// TwinCAT 3 PLC project Tc_EvenLogger
// Title: Tc_SystemServices
// Company: NewEngineer
// Author: https://github.com/phucpha
// ProjectVersion: 0.0.0.1
// Description: This library use for AlarmControler, Recipemanager,..
// ProgramVersion: 3.1.4024.0
// libraries:
//   Recipe Management, * (System)
//   Tc2_Standard, * (Beckhoff Automation GmbH)
//   Tc2_System, * (Beckhoff Automation GmbH)
//   Tc2_Utilities, * (Beckhoff Automation GmbH)
//   Tc3_EventLogger, * (Beckhoff Automation GmbH)
//   Tc3_Module, * (Beckhoff Automation GmbH)
//   TC3_Utilities_C, * (NewEngineer)
//   VisuDialogs, * (System)
//   VisuSymbols,3.5.10.0,System
// project tree:
//   DUTs/AlarmsEventLogger/AlarmControler/ E_AlarmControlerState.TcDUT (not stored)
//   DUTs/AlarmsEventLogger/VisuEvents/ E_EventType.TcDUT (not stored), ST_BaseEvent.TcDUT (not stored), ST_Event.TcDUT (not stored)
//   DUTs/Recipe Manager/ E_RecipesManagerReturns.TcDUT (not stored), E_RecipesManagerState.TcDUT (not stored), E_RecipesManagerStateBackup.TcDUT (not stored), E_RecipesManagerStateCreateRemove.TcDUT (not stored), E_RecipesManagerStateInit.TcDUT (not stored), E_RecipesManagerStateReload.TcDUT (not stored)
//   DUTs/Visus/AlarmControl/ E_VisuCtrlAlarmControlState.TcDUT (not stored)
//   DUTs/Visus/RecipeManager/ E_VisuCtrlRecipeParameterType.TcDUT (not stored), E_VisuCtrlRecipesManagerState.TcDUT (not stored), ST_VisuCtrlRecipeParameter.TcDUT (not stored), ST_VisuCtrlUnitFrame.TcDUT (not stored)
//   / GlobalTextList.TcGTLO, PlcTask.TcTTO, Visualization Manager.TcVMO (not stored)
//   GVLs/ GVL.TcGVL
//   POUs/AlarmsEventlogger/AlarmControler/ FB_AlarmControler.TcPOU (not stored), I_AlarmControler.TcIO (not stored)
//   POUs/AlarmsEventlogger/VisuEvents/ FB_VisuEventsHandling.TcPOU (not stored), LDT_TO_STRING.TcPOU (not stored)
//   POUs/Recipes Manager/ FB_RecipeParameter.TcPOU (not stored), FB_RecipesControler.TcPOU (not stored), I_RecipeParameter.TcIO (not stored), I_RecipesManager.TcIO (not stored)
//   VISUs/Alarms/ EventTable.TcVIS, EventTableNew.TcVIS (not stored), SingleEvent.TcVIS (not stored)
//   VISUs/Alarms/Image Pools/ IP_EventSeverity.TcIPO (not stored), IP_EventType.TcIPO (not stored)
//   VISUs/Alarms/Text Lists/ TL_EventServerity.TcTLO, TL_EventType.TcTLO (not stored)
//   VISUs/Pages/ PageAlarms.TcVIS (not stored), PageRecipesManager.TcVIS (not stored)
//   VISUs/Recipes/ SingleRecipesParameterTypeBool.TcVIS, SingleRecipesParameterTypeInteger.TcVIS (not stored), SingleRecipesParameterTypeReal.TcVIS, SingleRecipesParameterTypeString.TcVIS
//   VISUs/Recipes/Text Lists/ TL_RecipesManagerReturns.TcTLO (not stored), TL_RecipesManagerStatus.TcTLO (not stored)

CONFIGURATION Tc_EvenLogger
    RESOURCE PLC ON TwinCAT3
        TASK PlcTask(INTERVAL := T#10ms, PRIORITY := 20);
    END_RESOURCE
END_CONFIGURATION

// ---- GVLs/GVL.TcGVL
VAR_GLOBAL CONSTANT
	(* --- Alarm controler --- *)
	iMAX_DEFINITION_EVENTS					: UDINT := 512; 													(* Maximum size of active alarms table *)
	iMAX_EVENTS								: UDINT	:= 512; 													(* Maximum size of events table *) 
	
	(* --- Recipes manager --- *)
	iMAX_NUMBER_OF_RECIPES					: USINT 		:= 128;												(* Defines maximum number of recipes stored in recipe manager *)
	iMAX_NUMBER_OF_VARIABLES_IN_RECIPES		: USINT			:= 128;												(* Defines maximum number of parameters stored inside the recipe *)
	iMAX_RECIPE_NAME_LENGTH					: INT			:= 80;												(* Defines maximum length of the recipe name *)
END_VAR

// ---- GlobalTextList.TcGTLO
TEXTLIST GlobalTextList
  331 = '%d'
  890 = '%f'
  976 = '%s'
  2051 = '/'
  1711 = 'Active alarms:'
  1670 = 'Active critical alarms:'
  780 = 'Active errors:'
  700 = 'Active warnings:'
  813 = 'All active alarms:'
  300 = 'Backup'
  2292 = 'Backup and restore from external directory'
  1549 = 'Clear all'
  277 = 'Close'
  1047 = 'Create'
  2909 = 'Create new recipe:'
  2120 = 'Current value'
  1738 = 'Error: %s'
  1107 = 'Event history:'
  86 = 'Event ID'
  619 = 'Event Text'
  297 = 'Event Type'
  77 = 'Export to file'
  1263 = 'Load from file'
  1606 = 'Next'
  1645 = 'Number of:'
  1309 = 'Path:'
  1825 = 'Previous'
  690 = 'Recipe list:'
  1499 = 'Recipe name:'
  247 = 'Recipe parameters'
  2656 = 'Recipes Manager: %s'
  2097 = 'Reload'
  2954 = 'Remove'
  561 = 'Restore'
  2626 = 'Save in file'
  550 = 'Select'
  7 = 'Selected recipe value'
  1458 = 'Selected recipe:'
  536 = 'Severity'
  848 = 'Time Cleared'
  730 = 'Time Confirmed'
  9 = 'Time Raised'
END_TEXTLIST

// ---- VISUs/Alarms/EventTable.TcVIS
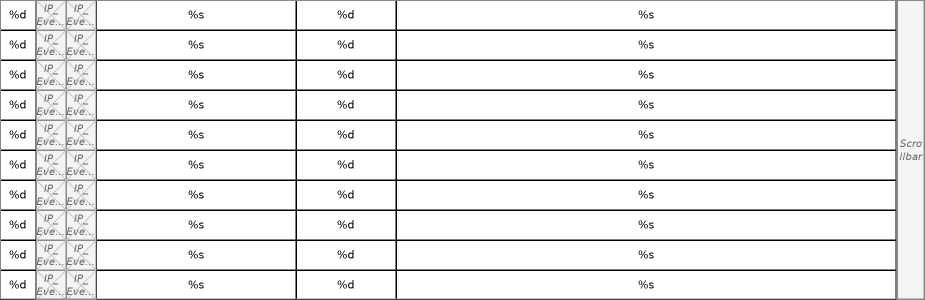
VISUALIZATION EventTable  // 925x300
VAR_IN_OUT
	data : ARRAY[1..512] OF ST_Event;
END_VAR
VAR 
	iIndex : INT;
END_VAR
    Group (0,0 896x30), invisible if: data[iIndex+1].iType = 0
        OnMouseClick: OpenDialog Dialog=SingleEvent, Parameters={data: data[iIndex+1]}, OpenModal=True, OpenCentered=True
        Rectangle (0,0 36x30), "%d", text variable: iIndex + 1
        Image (36,0 30x30), invisible if: data[iIndex+1].iType <> 1, image: IP_EventType.alarm
        Image (36,0 30x30), invisible if: data[iIndex+1].iType <> 2, image: IP_EventType.message
        Rectangle (96,0 200x30), "%s", text variable: LDT_TO_STRING(data[iIndex+1].iTimeStamp)
        Rectangle (296,0 100x30), "%d", text variable: data[iIndex+1].iEventId
        Image (66,0 30x30), invisible if: data[iIndex+1].eSeverity <> 4, image: IP_EventSeverity.critical
        Image (66,0 30x30), invisible if: data[iIndex+1].eSeverity <> 3, image: IP_EventSeverity.error
        Image (66,0 30x30), invisible if: data[iIndex+1].eSeverity <> 2, image: IP_EventSeverity.warning
        Image (66,0 30x30), invisible if: data[iIndex+1].eSeverity <> 1, image: IP_EventSeverity.info
        Image (66,0 30x30), invisible if: data[iIndex+1].eSeverity <> 0, image: IP_EventSeverity.verbose
        Rectangle (396,0 500x30), "%s", text variable: data[iIndex+1].sEventText
    Group (0,30 896x30), invisible if: data[iIndex+2].iType = 0
        OnMouseClick: OpenDialog Dialog=SingleEvent, Parameters={data: data[iIndex+2]}, OpenModal=True, OpenCentered=True
        Rectangle (0,0 36x30), "%d", text variable: iIndex + 2
        Image (36,0 30x30), invisible if: data[iIndex+2].iType <> 1, image: IP_EventType.alarm
        Image (36,0 30x30), invisible if: data[iIndex+2].iType <> 2, image: IP_EventType.message
        Rectangle (96,0 200x30), "%s", text variable: LDT_TO_STRING(data[iIndex+2].iTimeStamp)
        Rectangle (296,0 100x30), "%d", text variable: data[iIndex+2].iEventId
        Image (66,0 30x30), invisible if: data[iIndex+2].eSeverity <> 4, image: IP_EventSeverity.critical
        Image (66,0 30x30), invisible if: data[iIndex+2].eSeverity <> 3, image: IP_EventSeverity.error
        Image (66,0 30x30), invisible if: data[iIndex+2].eSeverity <> 2, image: IP_EventSeverity.warning
        Image (66,0 30x30), invisible if: data[iIndex+2].eSeverity <> 1, image: IP_EventSeverity.info
        Image (66,0 30x30), invisible if: data[iIndex+2].eSeverity <> 0, image: IP_EventSeverity.verbose
        Rectangle (396,0 500x30), "%s", text variable: data[iIndex+2].sEventText
    Group (0,60 896x30), invisible if: data[iIndex+3].iType = 0
        OnMouseClick: OpenDialog Dialog=SingleEvent, Parameters={data: data[iIndex+3]}, OpenModal=True, OpenCentered=True
        Rectangle (0,0 36x30), "%d", text variable: iIndex + 3
        Image (36,0 30x30), invisible if: data[iIndex+3].iType <> 1, image: IP_EventType.alarm
        Image (36,0 30x30), invisible if: data[iIndex+3].iType <> 2, image: IP_EventType.message
        Rectangle (96,0 200x30), "%s", text variable: LDT_TO_STRING(data[iIndex+3].iTimeStamp)
        Rectangle (296,0 100x30), "%d", text variable: data[iIndex+3].iEventId
        Image (66,0 30x30), invisible if: data[iIndex+3].eSeverity <> 4, image: IP_EventSeverity.critical
        Image (66,0 30x30), invisible if: data[iIndex+3].eSeverity <> 3, image: IP_EventSeverity.error
        Image (66,0 30x30), invisible if: data[iIndex+3].eSeverity <> 2, image: IP_EventSeverity.warning
        Image (66,0 30x30), invisible if: data[iIndex+3].eSeverity <> 1, image: IP_EventSeverity.info
        Image (66,0 30x30), invisible if: data[iIndex+3].eSeverity <> 0, image: IP_EventSeverity.verbose
        Rectangle (396,0 500x30), "%s", text variable: data[iIndex+3].sEventText
    Group (0,90 896x30), invisible if: data[iIndex+4].iType = 0
        OnMouseClick: OpenDialog Dialog=SingleEvent, Parameters={data: data[iIndex+4]}, OpenModal=True, OpenCentered=True
        Rectangle (0,0 36x30), "%d", text variable: iIndex + 4
        Image (36,0 30x30), invisible if: data[iIndex+4].iType <> 1, image: IP_EventType.alarm
        Image (36,0 30x30), invisible if: data[iIndex+4].iType <> 2, image: IP_EventType.message
        Rectangle (96,0 200x30), "%s", text variable: LDT_TO_STRING(data[iIndex+4].iTimeStamp)
        Rectangle (296,0 100x30), "%d", text variable: data[iIndex+4].iEventId
        Image (66,0 30x30), invisible if: data[iIndex+4].eSeverity <> 4, image: IP_EventSeverity.critical
        Image (66,0 30x30), invisible if: data[iIndex+4].eSeverity <> 3, image: IP_EventSeverity.error
        Image (66,0 30x30), invisible if: data[iIndex+4].eSeverity <> 2, image: IP_EventSeverity.warning
        Image (66,0 30x30), invisible if: data[iIndex+4].eSeverity <> 1, image: IP_EventSeverity.info
        Image (66,0 30x30), invisible if: data[iIndex+4].eSeverity <> 0, image: IP_EventSeverity.verbose
        Rectangle (396,0 500x30), "%s", text variable: data[iIndex+4].sEventText
    Group (0,120 896x30), invisible if: data[iIndex+5].iType = 0
        OnMouseClick: OpenDialog Dialog=SingleEvent, Parameters={data: data[iIndex+5]}, OpenModal=True, OpenCentered=True
        Rectangle (0,0 36x30), "%d", text variable: iIndex + 5
        Image (36,0 30x30), invisible if: data[iIndex+5].iType <> 1, image: IP_EventType.alarm
        Image (36,0 30x30), invisible if: data[iIndex+5].iType <> 2, image: IP_EventType.message
        Rectangle (96,0 200x30), "%s", text variable: LDT_TO_STRING(data[iIndex+5].iTimeStamp)
        Rectangle (296,0 100x30), "%d", text variable: data[iIndex+5].iEventId
        Image (66,0 30x30), invisible if: data[iIndex+5].eSeverity <> 4, image: IP_EventSeverity.critical
        Image (66,0 30x30), invisible if: data[iIndex+5].eSeverity <> 3, image: IP_EventSeverity.error
        Image (66,0 30x30), invisible if: data[iIndex+5].eSeverity <> 2, image: IP_EventSeverity.warning
        Image (66,0 30x30), invisible if: data[iIndex+5].eSeverity <> 1, image: IP_EventSeverity.info
        Image (66,0 30x30), invisible if: data[iIndex+5].eSeverity <> 0, image: IP_EventSeverity.verbose
        Rectangle (396,0 500x30), "%s", text variable: data[iIndex+5].sEventText
    Group (0,150 896x30), invisible if: data[iIndex+6].iType = 0
        OnMouseClick: OpenDialog Dialog=SingleEvent, Parameters={data: data[iIndex+6]}, OpenModal=True, OpenCentered=True
        Rectangle (0,0 36x30), "%d", text variable: iIndex + 6
        Image (36,0 30x30), invisible if: data[iIndex+6].iType <> 1, image: IP_EventType.alarm
        Image (36,0 30x30), invisible if: data[iIndex+6].iType <> 2, image: IP_EventType.message
        Rectangle (96,0 200x30), "%s", text variable: LDT_TO_STRING(data[iIndex+6].iTimeStamp)
        Rectangle (296,0 100x30), "%d", text variable: data[iIndex+6].iEventId
        Image (66,0 30x30), invisible if: data[iIndex+6].eSeverity <> 4, image: IP_EventSeverity.critical
        Image (66,0 30x30), invisible if: data[iIndex+6].eSeverity <> 3, image: IP_EventSeverity.error
        Image (66,0 30x30), invisible if: data[iIndex+6].eSeverity <> 2, image: IP_EventSeverity.warning
        Image (66,0 30x30), invisible if: data[iIndex+6].eSeverity <> 1, image: IP_EventSeverity.info
        Image (66,0 30x30), invisible if: data[iIndex+6].eSeverity <> 0, image: IP_EventSeverity.verbose
        Rectangle (396,0 500x30), "%s", text variable: data[iIndex+6].sEventText
    Group (0,180 896x30), invisible if: data[iIndex+7].iType = 0
        OnMouseClick: OpenDialog Dialog=SingleEvent, Parameters={data: data[iIndex+7]}, OpenModal=True, OpenCentered=True
        Rectangle (0,0 36x30), "%d", text variable: iIndex + 7
        Image (36,0 30x30), invisible if: data[iIndex+7].iType <> 1, image: IP_EventType.alarm
        Image (36,0 30x30), invisible if: data[iIndex+7].iType <> 2, image: IP_EventType.message
        Rectangle (96,0 200x30), "%s", text variable: LDT_TO_STRING(data[iIndex+7].iTimeStamp)
        Rectangle (296,0 100x30), "%d", text variable: data[iIndex+7].iEventId
        Image (66,0 30x30), invisible if: data[iIndex+7].eSeverity <> 4, image: IP_EventSeverity.critical
        Image (66,0 30x30), invisible if: data[iIndex+7].eSeverity <> 3, image: IP_EventSeverity.error
        Image (66,0 30x30), invisible if: data[iIndex+7].eSeverity <> 2, image: IP_EventSeverity.warning
        Image (66,0 30x30), invisible if: data[iIndex+7].eSeverity <> 1, image: IP_EventSeverity.info
        Image (66,0 30x30), invisible if: data[iIndex+7].eSeverity <> 0, image: IP_EventSeverity.verbose
        Rectangle (396,0 500x30), "%s", text variable: data[iIndex+7].sEventText
    Group (0,210 896x30), invisible if: data[iIndex+8].iType = 0
        OnMouseClick: OpenDialog Dialog=SingleEvent, Parameters={data: data[iIndex+8]}, OpenModal=True, OpenCentered=True
        Rectangle (0,0 36x30), "%d", text variable: iIndex + 8
        Image (36,0 30x30), invisible if: data[iIndex+8].iType <> 1, image: IP_EventType.alarm
        Image (36,0 30x30), invisible if: data[iIndex+8].iType <> 2, image: IP_EventType.message
        Rectangle (96,0 200x30), "%s", text variable: LDT_TO_STRING(data[iIndex+8].iTimeStamp)
        Rectangle (296,0 100x30), "%d", text variable: data[iIndex+8].iEventId
        Image (66,0 30x30), invisible if: data[iIndex+8].eSeverity <> 4, image: IP_EventSeverity.critical
        Image (66,0 30x30), invisible if: data[iIndex+8].eSeverity <> 3, image: IP_EventSeverity.error
        Image (66,0 30x30), invisible if: data[iIndex+8].eSeverity <> 2, image: IP_EventSeverity.warning
        Image (66,0 30x30), invisible if: data[iIndex+8].eSeverity <> 1, image: IP_EventSeverity.info
        Image (66,0 30x30), invisible if: data[iIndex+8].eSeverity <> 0, image: IP_EventSeverity.verbose
        Rectangle (396,0 500x30), "%s", text variable: data[iIndex+8].sEventText
    Group (0,240 896x30), invisible if: data[iIndex+9].iType = 0
        OnMouseClick: OpenDialog Dialog=SingleEvent, Parameters={data: data[iIndex+9]}, OpenModal=True, OpenCentered=True
        Rectangle (0,0 36x30), "%d", text variable: iIndex + 9
        Image (36,0 30x30), invisible if: data[iIndex+9].iType <> 1, image: IP_EventType.alarm
        Image (36,0 30x30), invisible if: data[iIndex+9].iType <> 2, image: IP_EventType.message
        Rectangle (96,0 200x30), "%s", text variable: LDT_TO_STRING(data[iIndex+9].iTimeStamp)
        Rectangle (296,0 100x30), "%d", text variable: data[iIndex+9].iEventId
        Image (66,0 30x30), invisible if: data[iIndex+9].eSeverity <> 4, image: IP_EventSeverity.critical
        Image (66,0 30x30), invisible if: data[iIndex+9].eSeverity <> 3, image: IP_EventSeverity.error
        Image (66,0 30x30), invisible if: data[iIndex+9].eSeverity <> 2, image: IP_EventSeverity.warning
        Image (66,0 30x30), invisible if: data[iIndex+9].eSeverity <> 1, image: IP_EventSeverity.info
        Image (66,0 30x30), invisible if: data[iIndex+9].eSeverity <> 0, image: IP_EventSeverity.verbose
        Rectangle (396,0 500x30), "%s", text variable: data[iIndex+9].sEventText
    Group (0,270 896x30), invisible if: data[iIndex+10].iType = 0
        OnMouseClick: OpenDialog Dialog=SingleEvent, Parameters={data: data[iIndex+10]}, OpenModal=True, OpenCentered=True
        Rectangle (0,0 36x30), "%d", text variable: iIndex + 10
        Image (36,0 30x30), invisible if: data[iIndex+10].iType <> 1, image: IP_EventType.alarm
        Image (36,0 30x30), invisible if: data[iIndex+10].iType <> 2, image: IP_EventType.message
        Rectangle (96,0 200x30), "%s", text variable: LDT_TO_STRING(data[iIndex+10].iTimeStamp)
        Rectangle (296,0 100x30), "%d", text variable: data[iIndex+10].iEventId
        Image (66,0 30x30), invisible if: data[iIndex+10].eSeverity <> 4, image: IP_EventSeverity.critical
        Image (66,0 30x30), invisible if: data[iIndex+10].eSeverity <> 3, image: IP_EventSeverity.error
        Image (66,0 30x30), invisible if: data[iIndex+10].eSeverity <> 2, image: IP_EventSeverity.warning
        Image (66,0 30x30), invisible if: data[iIndex+10].eSeverity <> 1, image: IP_EventSeverity.info
        Image (66,0 30x30), invisible if: data[iIndex+10].eSeverity <> 0, image: IP_EventSeverity.verbose
        Rectangle (396,0 500x30), "%s", text variable: data[iIndex+10].sEventText
    Scrollbar (897,0 28x300)
        p2245068023: GVL.iMAX_EVENTS - 10
        p1057716461: iIndex
END_VISUALIZATION

// ---- VISUs/Alarms/Text Lists/TL_EventServerity.TcTLO
TEXTLIST TL_EventServerity
  0 = 'Verbose'
  1 = 'Info'
  2 = 'Warning'
  3 = 'Error'
  4 = 'Critical'
   = ''
END_TEXTLIST

// ---- VISUs/Recipes/SingleRecipesParameterTypeBool.TcVIS
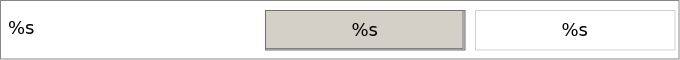
VISUALIZATION SingleRecipesParameterTypeBool  // 680x60
VAR_IN_OUT
	stRecipeParameter : ST_VisuCtrlRecipeParameter;
END_VAR
    Textfield (475,10 200x40), "%s", text variable: stRecipeParameter.sFileValue
    Textfield (5,8 250x40), "%s", text variable: stRecipeParameter.sName
    Button (265,10 200x40), "%s", text variable: stRecipeParameter.sName
        toggle stRecipeParameter.bValue
END_VISUALIZATION

// ---- VISUs/Recipes/SingleRecipesParameterTypeReal.TcVIS
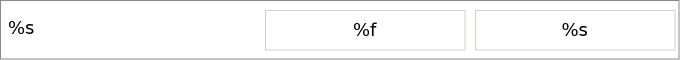
VISUALIZATION SingleRecipesParameterTypeReal  // 680x60
VAR_IN_OUT
	stRecipeParameter : ST_VisuCtrlRecipeParameter;
END_VAR
    Textfield (265,10 200x40), "%f", text variable: stRecipeParameter.rValue
        OnMouseClick: write the text variable via VisuDialogs.Numpad
    Textfield (475,10 200x40), "%s", text variable: stRecipeParameter.sFileValue
    Textfield (5,8 250x40), "%s", text variable: stRecipeParameter.sName
END_VISUALIZATION

// ---- VISUs/Recipes/SingleRecipesParameterTypeString.TcVIS
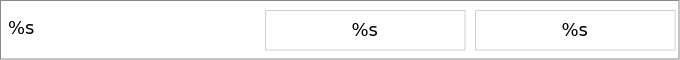
VISUALIZATION SingleRecipesParameterTypeString  // 680x60
VAR_IN_OUT
	stRecipeParameter : ST_VisuCtrlRecipeParameter;
END_VAR
    Textfield (265,10 200x40), "%s", text variable: stRecipeParameter.sValue
        OnMouseClick: write the text variable via VisuDialogs.Keypad
    Textfield (475,10 200x40), "%s", text variable: stRecipeParameter.sFileValue
    Textfield (5,8 250x40), "%s", text variable: stRecipeParameter.sName
END_VISUALIZATION
